(* PLC project DesignSpecificationDCMotorModel, Dassault Systèmes orchideo | easySSP (eXXcellent solutions GmbH) orchideo | easySSP (eXXcellent solutions GmbH) *)
(* stored: creationDateTime 2022-04-20T15:01:31Z, contentDescription extra/org.ssp-standard.ssp-traceability.stmd/Design-Specification-DC-Motor-Model_1.ssd *)

FUNCTION_BLOCK stimuli_model
  VAR_OUTPUT
    U : REAL := 0.0;
    M_load : REAL := 0.0;
  END_VAR


ACTION C_source_code:

END_ACTION
END_FUNCTION_BLOCK

FUNCTION_BLOCK edrive_mass_spec
  VAR_INPUT
    M_B : REAL := 0.0;
    M_A : REAL := 0.0;
  END_VAR
  VAR_OUTPUT
    phiA : REAL := 0.0;
    wB : REAL := 0.0;
    wA : REAL := 0.0;
    phiB : REAL := 0.0;
  END_VAR


ACTION C_source_code:

END_ACTION
END_FUNCTION_BLOCK

FUNCTION_BLOCK emachine_model
  VAR_INPUT
    w : REAL := 0.0;
    U : REAL := 0.0;
    phi : REAL := 0.0;
  END_VAR
  VAR_OUTPUT
    M : REAL := 0.0;
    I : REAL := 0.0;
  END_VAR


ACTION C_source_code:

END_ACTION
END_FUNCTION_BLOCK

PROGRAM SuT
  VAR_INPUT
    M_load : REAL := 0.0;
    U : REAL := 0.0;
  END_VAR
  VAR_OUTPUT
    M_mot : REAL := 0.0;
    phiB : REAL := 0.0;
    wB : REAL := 0.0;
    I : REAL := 0.0;
  END_VAR

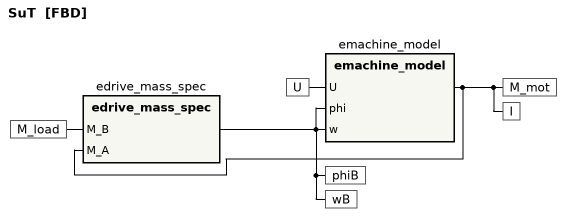
(* FBD diagram, written out as Structured Text *)
edrive_mass_spec(M_B := M_load, M_A := emachine_model.M);
emachine_model(U := U, phi := edrive_mass_spec.phiA, w := edrive_mass_spec.wA);
M_mot := emachine_model.M;
phiB := edrive_mass_spec.phiB;
wB := edrive_mass_spec.wB;
I := emachine_model.I;
END_PROGRAM

PROGRAM DesignSpecificationDCMotorModel.DesignSpecificationDCMotorModel
  VAR_OUTPUT
    wB : REAL := 0.0;
    U : REAL := 0.0;
    M_mot : REAL := 0.0;
    I : REAL := 0.0;
  END_VAR

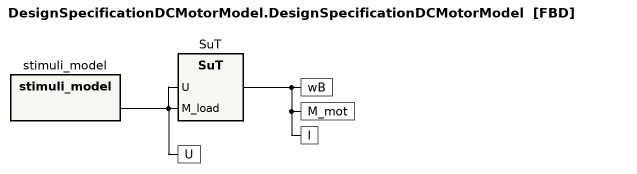
(* FBD diagram, written out as Structured Text *)
stimuli_model();
SuT(U := stimuli_model.U, M_load := stimuli_model.M_load);
wB := SuT.wB;
U := stimuli_model.U;
M_mot := SuT.M_mot;
I := SuT.I;
END_PROGRAM
